% RSLogix 500 project TRAFFIC LIGHT SEQUENCER.RSS, saved by version 8.30.00.16 %
PROJECT "UNTITLED"    % processor: MicroLogix 1000 %

PROGRAM FILES
  LAD 2 "MAIN_PROG"  9 rungs
  LAD 3 "FLASHER"  4 rungs
  LAD 4 "TIMER"  5 rungs
  LAD 5 "STI_INT"  1 rungs
  LAD 6, 7, 8, 9, 10, 11, 12, 13, 14, 15, 16: only END

DATA FILES
  O0 OUTPUT  1 elements
  I1 INPUT  2 elements
  S2 STATUS  33 elements
  B3 BINARY  32 elements
  T4 TIMER  40 elements
  C5 COUNTER  32 elements
  R6 CONTROL  16 elements
  N7 INTEGER  105 elements

LADDER 2 "MAIN_PROG"
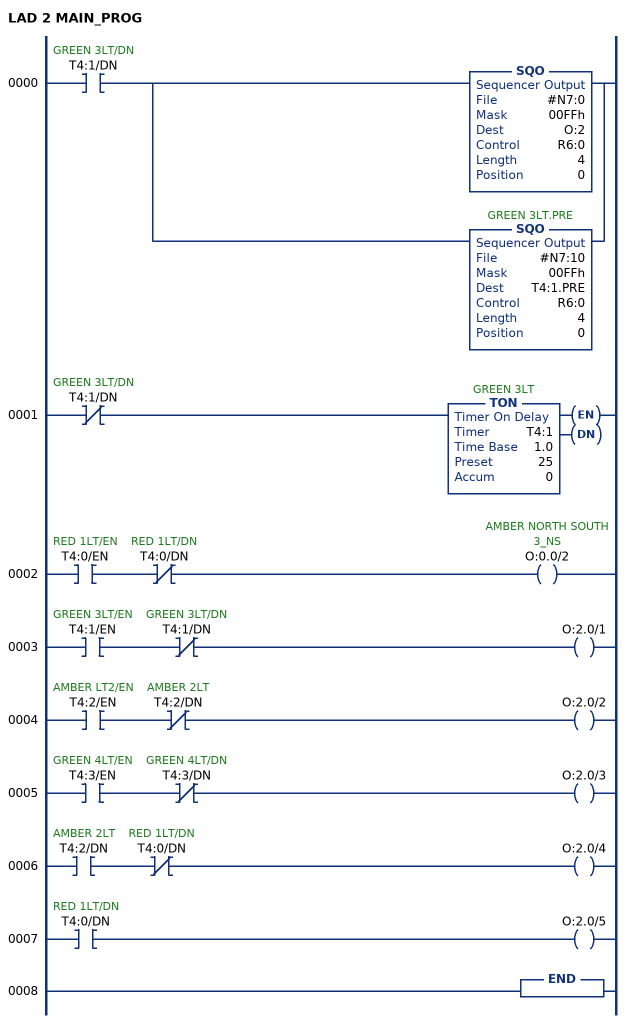
% Rung: 0 %  % edit flag set %
SOR XIC T4:1/DN BST SQO #N7:0 00FFh O:2 R6:0 4 0 NXB SQO #N7:10 00FFh T4:1.PRE R6:0 4 0 BND EOR
%   T4:1  3LT  "GREEN" %
%   N7:0  N7 %
% Rung: 1 %
SOR XIO T4:1/DN TON T4:1 1.0 25 0 EOR
%   T4:1  3LT  "GREEN" %
% Rung: 2 %
SOR XIC T4:0/EN XIO T4:0/DN OTE O:0.0/2 EOR
%   T4:0  1LT  "RED" %
%   O:0.0/2  3_NS  "AMBER NORTH SOUTH" %
% Rung: 3 %  % edit flag set %
SOR XIC T4:1/EN XIO T4:1/DN OTE O:2.0/1 EOR
%   T4:1  3LT  "GREEN" %
% Rung: 4 %  % edit flag set %
SOR XIC T4:2/EN XIO T4:2/DN OTE O:2.0/2 EOR
%   T4:2  LT2  "AMBER" %
%   T4:2/DN  2LT  "AMBER" %
% Rung: 5 %  % edit flag set %
SOR XIC T4:3/EN XIO T4:3/DN OTE O:2.0/3 EOR
%   T4:3  4LT  "GREEN" %
% Rung: 6 %  % edit flag set %
SOR XIC T4:2/DN XIO T4:0/DN OTE O:2.0/4 EOR
%   T4:2/DN  2LT  "AMBER" %
%   T4:0  1LT  "RED" %
% Rung: 7 %  % edit flag set %
SOR XIC T4:0/DN OTE O:2.0/5 EOR
%   T4:0  1LT  "RED" %
% Rung: 8 %
SOR END EOR

LADDER 3 "FLASHER"
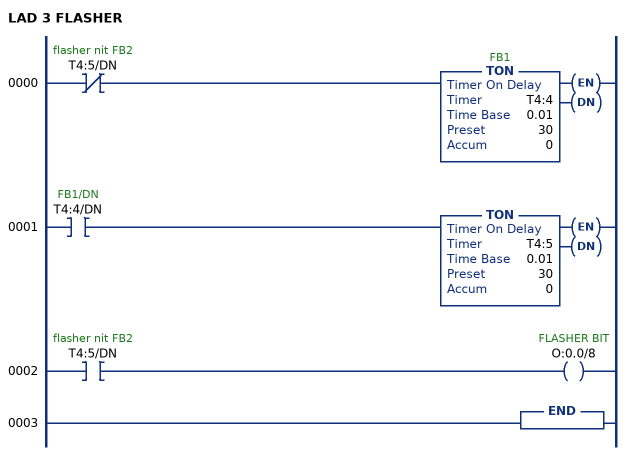
% Rung: 0 %
SOR XIO T4:5/DN TON T4:4 0.01 30 0 EOR
%   T4:5/DN  FB2  "flasher nit" %
%   T4:4  FB1 %
% Rung: 1 %
SOR XIC T4:4/DN TON T4:5 0.01 30 0 EOR
%   T4:4  FB1 %
% Rung: 2 %
SOR XIC T4:5/DN OTE O:0.0/8 EOR
%   T4:5/DN  FB2  "flasher nit" %
%   O:0.0/8  "FLASHER BIT" %
% Rung: 3 %
SOR END EOR

LADDER 4 "TIMER"
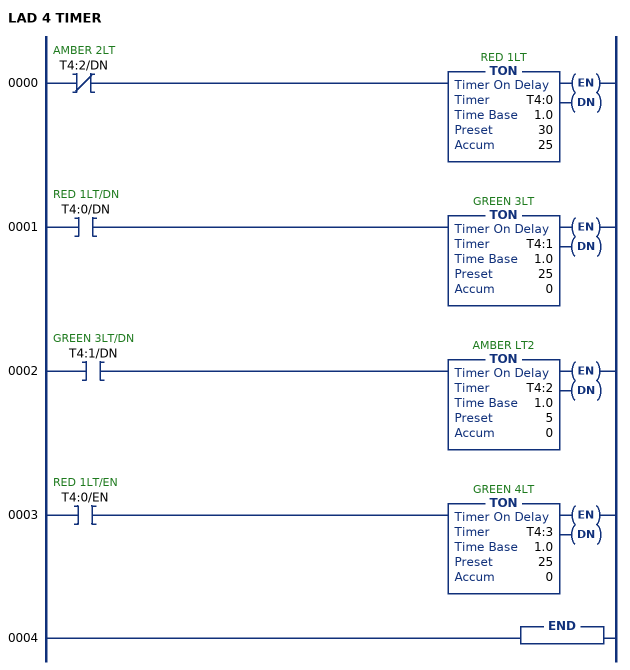
% Rung: 0 %
SOR XIO T4:2/DN TON T4:0 1.0 30 25 EOR
%   T4:2/DN  2LT  "AMBER" %
%   T4:0  1LT  "RED" %
% Rung: 1 %
SOR XIC T4:0/DN TON T4:1 1.0 25 0 EOR
%   T4:0  1LT  "RED" %
%   T4:1  3LT  "GREEN" %
% Rung: 2 %
SOR XIC T4:1/DN TON T4:2 1.0 5 0 EOR
%   T4:1  3LT  "GREEN" %
%   T4:2  LT2  "AMBER" %
% Rung: 3 %
SOR XIC T4:0/EN TON T4:3 1.0 25 0 EOR
%   T4:0  1LT  "RED" %
%   T4:3  4LT  "GREEN" %
% Rung: 4 %
SOR END EOR

OTHER DOCUMENTED ADDRESSES
  B3:0/0  FB  "FLASHER BIT"
  O:0.0/0  1_NS  "RED NORTH SOUTH"
  O:0.0/1  2_NS  "GREEN NORTH SOUTH"
  O:0.0/3  4_NS  "WALK NORTH SOUTH"
  O:0.0/4  1_EW  "GREEN EAST WEST"
  O:0.0/5  3EW  "AMBER EAST WEST"
  O:0.0/6  3_EW  "RED EAST WEST"
  O:0.0/7  4_EW  "WALK EAST WEST"

DATA TABLE (non-zero values as saved)
DATA T4
% .PRE .ACC %
% T4:0 % 30 25
% T4:1 % 25 0
% T4:2 % 5 0
% T4:3 % 25 0
% T4:4 % 30 0
% T4:5 % 30 0
DATA R6
% .LEN .POS %
% R6:0 % 4 0
DATA N7
% N7:10 % 1 0 0 0 0 0 1 0 0 0
% N7:20 % 1 0 0 0 0 1 0 0 0 0
% N7:30 % 0 0 1 0 1 0 0 0 0 0
% N7:40 % 0 1 0 0 1 0 0 0 0 0
